// TIA Portal V20 export
FUNCTION "IO Mapping" : Void   // FC100, LAD
{ S7_Optimized_Access := 'TRUE' }
// stored: SetENOAutomatically false
   VAR_INPUT
      sensor1 : Bool;
      sensor2 : Bool;
      sensor3 : Bool;
      sensor4 : Bool;
      sensor5 : Bool;
      sensor6 : Bool;
      sensor7 : Bool;
      sensor8 : Bool;
      sensor9 : Bool;
      sensor10 : Bool;
   END_VAR
   VAR_OUTPUT
      O_sensor1 : Bool;
      O_sensor2 : Bool;
      O_sensor3 : Bool;
      O_sensor4 : Bool;
      O_sensor5 : Bool;
      O_sensor6 : Bool;
      O_sensor7 : Bool;
      O_sensor8 : Bool;
      O_sensor9 : Bool;
      O_sensor10 : Bool;
   END_VAR
BEGIN

REGION Network 1
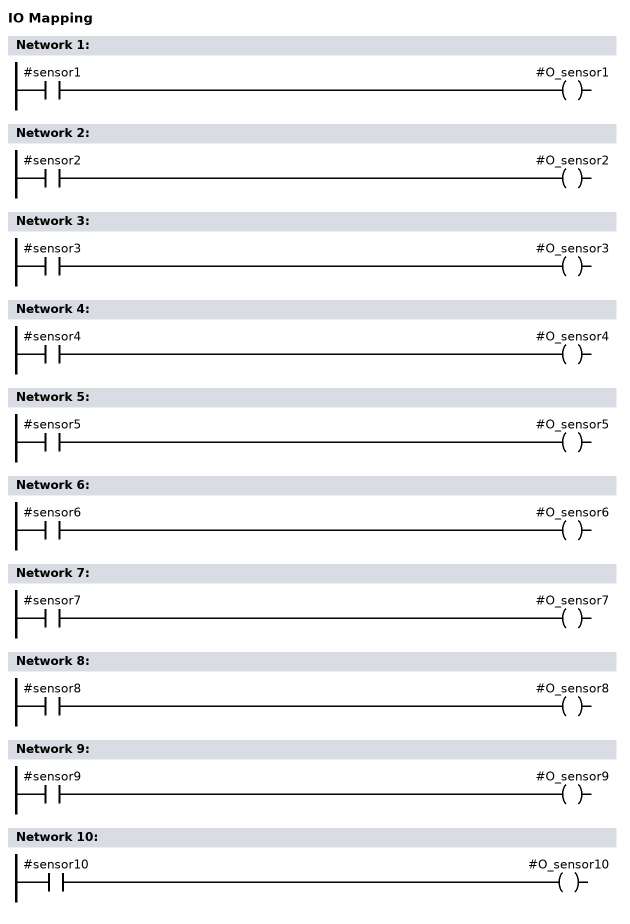
   RUNG wire#powerrail
      Contact( #sensor1 )
      Coil( #O_sensor1 )
   END_RUNG
   // the same network as SCL:
   #O_sensor1 := #sensor1;
END_REGION

REGION Network 2
   RUNG wire#powerrail
      Contact( #sensor2 )
      Coil( #O_sensor2 )
   END_RUNG
   // the same network as SCL:
   #O_sensor2 := #sensor2;
END_REGION

REGION Network 3
   RUNG wire#powerrail
      Contact( #sensor3 )
      Coil( #O_sensor3 )
   END_RUNG
   // the same network as SCL:
   #O_sensor3 := #sensor3;
END_REGION

REGION Network 4
   RUNG wire#powerrail
      Contact( #sensor4 )
      Coil( #O_sensor4 )
   END_RUNG
   // the same network as SCL:
   #O_sensor4 := #sensor4;
END_REGION

REGION Network 5
   RUNG wire#powerrail
      Contact( #sensor5 )
      Coil( #O_sensor5 )
   END_RUNG
   // the same network as SCL:
   #O_sensor5 := #sensor5;
END_REGION

REGION Network 6
   RUNG wire#powerrail
      Contact( #sensor6 )
      Coil( #O_sensor6 )
   END_RUNG
   // the same network as SCL:
   #O_sensor6 := #sensor6;
END_REGION

REGION Network 7
   RUNG wire#powerrail
      Contact( #sensor7 )
      Coil( #O_sensor7 )
   END_RUNG
   // the same network as SCL:
   #O_sensor7 := #sensor7;
END_REGION

REGION Network 8
   RUNG wire#powerrail
      Contact( #sensor8 )
      Coil( #O_sensor8 )
   END_RUNG
   // the same network as SCL:
   #O_sensor8 := #sensor8;
END_REGION

REGION Network 9
   RUNG wire#powerrail
      Contact( #sensor9 )
      Coil( #O_sensor9 )
   END_RUNG
   // the same network as SCL:
   #O_sensor9 := #sensor9;
END_REGION

REGION Network 10
   RUNG wire#powerrail
      Contact( #sensor10 )
      Coil( #O_sensor10 )
   END_RUNG
   // the same network as SCL:
   #O_sensor10 := #sensor10;
END_REGION
END_FUNCTION
